Staubli VAL3: changePoint.pgx

program changePoint(num x_nIndex)
  local num i
  local string l_sMessage[3]
  local num l_nLocal
  local bool l_bOk
  local num l_nStop
  local string l_sButton[2]
  local string l_sEmpty
  local string l_sItem
  local string l_sData
  local string l_sPath
begin

end
